FUNCTION_BLOCK SK_Tare (* Skill primitive Tare: Tare the scale (parameters: none). OPC UA Start(Session, parameters...)/Stop/Abort/Reset(Session) -> [Accepted, ErrorID]; START/HALT/ABORT/RESET from a parent -> SUCCESS or FAILURE(ErrorID) *)
  (* Standard: 61499-2 *)
  (* Version 0.1, 2026-09-28, Project contributors, AAU Smart Production Lab *)
  PACKAGE filling;
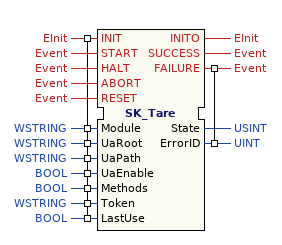
  EVENT_INPUT
    INIT : EInit WITH Module, UaRoot, UaPath, UaEnable, Methods, Token, LastUse;
    START;
    HALT;
    ABORT;
    RESET;
  END_EVENT
  EVENT_OUTPUT
    INITO : EInit;
    SUCCESS;
    FAILURE WITH ErrorID;
  END_EVENT
  VAR_INPUT
    Module : WSTRING;
    UaRoot : WSTRING;
    UaPath : WSTRING;
    UaEnable : BOOL;
    Methods : BOOL;
    Token : WSTRING;
    LastUse : BOOL := TRUE;
  END_VAR
  VAR_OUTPUT
    State : USINT;
    ErrorID : UINT;
  END_VAR
  FBS
    Control : modlib::SKILL_Control(InRange := TRUE);
    Owner : modlib::MOD_OwnerView;
    Mode : modlib::MOD_StateView;
    UaStart : iec61499::net::SERVER_2_1;
    UaStop : iec61499::net::SERVER_2_1;
    UaAbort : iec61499::net::SERVER_2_1;
    UaReset : iec61499::net::SERVER_2_1;
    PubState : iec61499::net::PUBLISH_2;
    Act : iec61499::net::PUBLISH_1(QI := TRUE);
    Logic : filling::SL_Tare(Equipment := "Scale");
    EqState : iec61499::net::SUBSCRIBE_2(QI := TRUE);
    EqView : filling::EV_Scale;
    WaitT : iec61499::events::E_DELAY(DT := T#500ms);
    EqCmd : iec61499::net::PUBLISH_4(QI := TRUE);
    Timer : iec61499::events::E_DELAY;
  END_FBS
  EVENT_CONNECTIONS
    Control.RSP_START TO UaStart.RSP;
    Control.RSP_STOP TO UaStop.RSP;
    Control.RSP_ABORT TO UaAbort.RSP;
    Control.RSP_RESET TO UaReset.RSP;
    UaStop.IND TO Control.CMD_STOP;
    UaAbort.IND TO Control.CMD_ABORT;
    UaReset.IND TO Control.CMD_RESET;
    UaStart.IND TO Control.CMD_START;
    Owner.CHG TO Control.OWNER_CHG;
    Mode.CHG TO Control.MOD_CHG;
    Control.PUB TO PubState.REQ;
    Control.ACT TO Act.REQ;
    START TO Control.START;
    HALT TO Control.HALT;
    ABORT TO Control.ABORT;
    RESET TO Control.RESET;
    Control.SUCCESS TO SUCCESS;
    Control.FAILURE TO FAILURE;
    INIT TO Control.INIT;
    Control.INITO TO Logic.INIT;
    Logic.INITO TO Owner.INIT;
    Owner.INITO TO Mode.INIT;
    Mode.INITO TO UaStart.INIT;
    UaStart.INITO TO UaStop.INIT;
    UaStop.INITO TO UaAbort.INIT;
    UaAbort.INITO TO UaReset.INIT;
    UaReset.INITO TO PubState.INIT;
    PubState.INITO TO Act.INIT;
    Act.INITO TO EqState.INIT;
    EqState.INITO TO EqCmd.INIT;
    EqCmd.INITO TO PubState.REQ;
    EqCmd.INITO TO INITO;
    Control.GO_UA TO Logic.START;
    Control.GO_PARENT TO Logic.START;
    Control.HALT_O TO Logic.HALT;
    Control.ABORT_O TO Logic.ABORT;
    Control.RUN_STOP TO Control.STOP_DONE;
    Logic.DONE TO Control.EXEC_DONE;
    Logic.FAILED TO Control.EXEC_FAILED;
    Logic.HALTED TO Control.EXEC_FAILED;
    EqState.IND TO EqView.REQ;
    EqView.CNF TO Logic.SAMPLE;
    Logic.CMD TO EqCmd.REQ;
    Logic.WAIT_START TO WaitT.START;
    Logic.WAIT_STOP TO WaitT.STOP;
    WaitT.EO TO Logic.WAIT_OVER;
    Logic.TIMER_START TO Timer.START;
    Logic.TIMER_STOP TO Timer.STOP;
    Timer.EO TO Logic.TIMER;
  END_CONNECTIONS
  DATA_CONNECTIONS
    Module TO Control.Module;
    Module TO Owner.Module;
    Module TO Mode.Module;
    UaRoot TO Control.UaRoot;
    UaPath TO Control.UaPath;
    Methods TO UaStart.QI;
    Methods TO UaStop.QI;
    Methods TO UaAbort.QI;
    Methods TO UaReset.QI;
    UaEnable TO PubState.QI;
    Control.IdStart TO UaStart.ID;
    Control.Accepted TO UaStart.SD_1;
    Control.RspError TO UaStart.SD_2;
    UaStart.RD_1 TO Control.S_Start;
    Control.IdStop TO UaStop.ID;
    Control.Accepted TO UaStop.SD_1;
    Control.RspError TO UaStop.SD_2;
    UaStop.RD_1 TO Control.S_Stop;
    Control.IdAbort TO UaAbort.ID;
    Control.Accepted TO UaAbort.SD_1;
    Control.RspError TO UaAbort.SD_2;
    UaAbort.RD_1 TO Control.S_Abort;
    Control.IdReset TO UaReset.ID;
    Control.Accepted TO UaReset.SD_1;
    Control.RspError TO UaReset.SD_2;
    UaReset.RD_1 TO Control.S_Reset;
    Owner.Owner TO Control.Owner;
    Mode.State TO Control.ModState;
    Control.IdPub TO PubState.ID;
    Control.State TO PubState.SD_1;
    Control.State TO State;
    Control.ErrorID TO PubState.SD_2;
    Control.ErrorID TO ErrorID;
    Control.IdAct TO Act.ID;
    Control.Delta TO Act.SD_1;
    Module TO Logic.Module;
    Token TO Logic.Token;
    LastUse TO Logic.LastUse;
    Logic.ErrorID TO Control.ExecError;
    Logic.EqFree TO Control.EqFree;
    Logic.IdEqState TO EqState.ID;
    EqState.RD_1 TO EqView.I_Weight;
    EqState.RD_2 TO EqView.I_Holder;
    EqView.Holder TO Logic.Holder;
    Logic.IdEqCmd TO EqCmd.ID;
    Logic.C_Holder TO EqCmd.SD_1;
    Logic.C_Command TO EqCmd.SD_2;
    Logic.C_Arg TO EqCmd.SD_3;
    Logic.C_Release TO EqCmd.SD_4;
    Logic.TimerDT TO Timer.DT;
  END_CONNECTIONS
END_FUNCTION_BLOCK
